FUNCTION_BLOCK FB_1s_UPS_BAPI EXTENDS FB_1s_UPS_Base
VAR CONSTANT
	nOkCapacityLevel	:BYTE	:=90;
END_VAR
VAR
	fb1sUps				:FB_S_UPS_BAPI;
END_VAR

METHOD Execute
fb1sUps(sNetID				:=F_CreateAmsNetId(_PcAmsNetId),
		iPLCPort			:=TwinCAT_SystemInfoVarList._AppInfo.AdsPort,
		tTimeout			:=DEFAULT_ADS_TIMEOUT,
		eUpsMode			:=E_S_UPS_Mode.eSUPS_WrPersistData_Shutdown,
		ePersistentMode		:=E_PersistentMode.SPDM_2PASS,
		tRecoverTime		:=T#10S,
		bPowerFailDetect	=>,
		eState				=>SUPER^._e1sUpsState,
		nCapacity			=>,
		bBusy				=>,
		bError				=>,
		nErrID				=>
		);
		
IF fb1sUps.bPowerFailDetect THEN
	SUPER^._bPowerFailDetect:=TRUE;
END_IF

SUPER^._bReady:=(fb1sUps.eState=E_S_UPS_State.eSUPS_PowerOK) AND (nOkCapacityLevel<fb1sUps.nCapacity) AND (fb1sUps.bError=FALSE);
END_METHOD

END_FUNCTION_BLOCK

(* stored: Version 1.1.0.1
   POU FB_1s_UPS_BAPI: Id {0be639e9-85f4-4d15-a6ba-bebd7c0856d3}, SpecialFunc None
   Method Execute: Id {3a7e3fc0-6360-4943-bda6-d23d23697136} *)
